{attribute 'no_check'}
//Convert a time value into a Lreal value in <s.ms> 
FUNCTION TIME_TO_FMRLREAL : LREAL
VAR_INPUT
	TIME_IN													:	TIME;
	NoOfDigits												:   INT(0..10) := 0; (* amount of decimaldigis*)
END_VAR             										
VAR                     									
	X														:	LREAL;
END_VAR

TIME_TO_FMRLREAL 											:= TIME_TO_LREAL(TIME_IN) ;
IF NoOfDigits > 0
THEN
	X														:= EXPT(10.0,ABS( NoOfDigits));
	TIME_TO_FMRLREAL										:= TIME_TO_FMRLREAL / X;
END_IF

END_FUNCTION

(* stored: Version 1.1.0.1, ProductVersion 3.1.4024.2
   POU TIME_TO_FMRLREAL: Id {f05ddee0-3dd8-4cf9-9849-b1322c227de1}, SpecialFunc None *)
